{attribute 'GeneratedUsingTerminal: EK1100-0000-0018'}
{attribute addProperty BoxType "EK1100-0000-0018"}
{attribute addProperty Id "Beckhoff_EJ9xxxEK1122Beckhoff_EJ9xxxEK1122_C80E1DB32A_0001_EJ9001_0000_0016EJ9001_1FC0878B2A_0002_EJ9505_0000_0016EJ9505_19A4723D6A_0003_EJ9576_0000_0018EJ9576_6D7359CA28A_0004_EJ9576_0000_0019EJ9576_85AB580429A_0005_EJ9576_0000_0020EJ9576_1017F4A528A_0006_EJ9576_0000_0022EJ9576_C42142C629"}
{attribute addProperty CRC "1226815735"}
{attribute addProperty Size "124"}
TYPE Beckhoff_EJ9xxx_491FB8F7 EXTENDS EK1100_1FC0878B :
STRUCT
	{attribute addProperty Name "Beckhoff_EJ9xxxEK1122"}
	{attribute addProperty PreviousPort "Beckhoff EJ9xxx : B"}
	Beckhoff_EJ9xxxEK1122 : Beckhoff_EJ9xxxEK1122_C80E1DB3;
	{attribute addProperty Name "A_0001_EJ9001_0000_0016"}
	{attribute addProperty PreviousPort "Beckhoff EJ9xxxEK1122 : C"}
	A_0001_EJ9001_0000_0016 : EJ9001_1FC0878B;
	{attribute addProperty Name "A_0002_EJ9505_0000_0016"}
	{attribute addProperty PreviousPort "A_0001(EJ9001-0000-0016) : B"}
	A_0002_EJ9505_0000_0016 : EJ9505_19A4723D;
	{attribute addProperty Name "A_0003_EJ9576_0000_0018"}
	{attribute addProperty PreviousPort "A_0002(EJ9505-0000-0016) : B"}
	A_0003_EJ9576_0000_0018 : EJ9576_6D7359CA;
	{attribute addProperty Name "A_0004_EJ9576_0000_0019"}
	{attribute addProperty PreviousPort "A_0003(EJ9576-0000-0018) : B"}
	A_0004_EJ9576_0000_0019 : EJ9576_85AB5804;
	{attribute addProperty Name "A_0005_EJ9576_0000_0020"}
	{attribute addProperty PreviousPort "A_0004(EJ9576-0000-0019) : B"}
	A_0005_EJ9576_0000_0020 : EJ9576_1017F4A5;
	{attribute addProperty Name "A_0006_EJ9576_0000_0022"}
	{attribute addProperty PreviousPort "A_0005(EJ9576-0000-0020) : B"}
	A_0006_EJ9576_0000_0022 : EJ9576_C42142C6;
END_STRUCT
END_TYPE

(* stored: Version 1.2.0.0, ProductVersion 3.1.4024.9
   DUT Beckhoff_EJ9xxx_491FB8F7: Id {928c934c-8727-42b3-a438-e66f7678b619} *)
